# EPICS autosave request: mcaApp/Db/SIS38XX_settings.req
$(P)PresetReal
$(P)Dwell
$(P)Prescale
$(P)ChannelAdvance
$(P)CountOnStart
$(P)Channel1Source
$(P)ReadAll.SCAN
$(P)NuseAll
$(P)EnableClientWait
$(P)MUXOutput
$(P)UserLED
$(P)InputMode
$(P)OutputMode
$(P)OutputPolarity
$(P)LNEStretcherEnable
$(P)LNEOutputPolarity
$(P)LNEOutputWidth
$(P)LNEOutputDelay
